(* PLC project CoDeSys External Library Template, WAGO e!COCKPIT e!COCKPIT, author 3S - Smart Software Solutions GmbH *)
(* stored: creationDateTime 2019-10-29T12:22:40.3197062, version 3.5.5.30, modificationDateTime 2019-10-24T14:40:07.960949, organization 3S - Smart Software Solutions GmbH *)
(* Library project template with all possible element types, docu and a sample project structure *)

(* values of enumModbusKodyFunkcji: OdczytWyjscBitowych: odczyt stanu wyjść cyfrowych; OdczytWejscBitowych: odczyt stanu wejść cyfrowych; OdczytNRejestrow: odczyt dowolnej ilości rejestrów; OdczytNRejestrowWejsciowych: odczyt dowolnej ilości rejestrów wejściowych; ZapisBitu: zapis jednego bitu informacji; ZapisRejestru: zapis jednego rejestru; OdczytStatusu: odczyt statusu; ZapisNBitow: zapis dowolnej ilości bitów; ZapisNRejestrow: zapis dowolnej ilości rejestrów *)

(* Nazwa bloku: Enumeracja - definicja kodów funkcyjnych protokołu modbus Projekt: Bałtyckie Centrum Biznesu Budynek 2 Firma: Solwena Autor: Marcin Szumiło Wersja: 0.1.0.1 - 2017-01-10 *)
{attribute 'qualified_only'}
{attribute 'strict'}
TYPE enumModbusKodyFunkcji : (OdczytWyjscBitowych := 1, OdczytWejscBitowych := 2, OdczytNRejestrow := 3, OdczytNRejestrowWejsciowych := 4, ZapisBitu := 5, ZapisRejestru := 6, OdczytStatusu := 7, ZapisNBitow := 15, ZapisNRejestrow := 16);
END_TYPE
